{attribute addProperty BoxType "KL8610-0004"}
{attribute addProperty Id "KL8601_1KL_B0A8062F00KL8601_2KL_B0A8062F00KL8601_3KL_B0A8062F00KL8601_4KL_B0A8062F00KL8601_5KL_B0A8062F00"}
{attribute addProperty CRC "2164849454"}
{attribute addProperty SizeInBites "0"}
{attribute addProperty SizeInBytes "0"}
TYPE KL_8108FB2E :
STRUCT
	{attribute addProperty Name "KL8601_1"}
	KL8601_1 : KL_B0A8062F;
	{attribute addProperty Name "KL8601_2"}
	KL8601_2 : KL_B0A8062F;
	{attribute addProperty Name "KL8601_3"}
	KL8601_3 : KL_B0A8062F;
	{attribute addProperty Name "KL8601_4"}
	KL8601_4 : KL_B0A8062F;
	{attribute addProperty Name "KL8601_5"}
	KL8601_5 : KL_B0A8062F;
END_STRUCT
END_TYPE

(* stored: Version 1.2.0.0, ProductVersion 3.1.4024.9
   DUT KL_8108FB2E: Id {66fc97ca-940c-4b34-89b8-4bb3eed9824f} *)
